PROGRAM PRG_IM2K4_PPM
VAR
    {attribute 'pytmc' := '
        pv: IM2K4:PPM
        io: io
    '}
    {attribute 'TcLinkTo' := '.fbGige.iIlluminatorINT := TIIB[IM2K4-EL4004-E7]^AO Outputs Channel 1^Analog output;
                              .fbGige.bGigePower := TIIB[IM2K4-EL2004-E3]^Channel 2^Output;
                              .fbPowerMeter.iVoltageINT := TIIB[IM2K4-EL3062-E6]^AI Standard Channel 1^Value;
                              .fbPowerMeter.fbThermoCouple.bError := TIIB[IM2K4-EL3314-E4]^TC Inputs Channel 1^Status^Error;
                              .fbPowerMeter.fbThermoCouple.bUnderrange := TIIB[IM2K4-EL3314-E4]^TC Inputs Channel 1^Status^Underrange;
                              .fbPowerMeter.fbThermoCouple.bOverrange := TIIB[IM2K4-EL3314-E4]^TC Inputs Channel 1^Status^Overrange;
                              .fbPowerMeter.fbThermoCouple.iRaw := TIIB[IM2K4-EL3314-E4]^TC Inputs Channel 1^Value;
                              .fbYagThermoCouple.bError := TIIB[IM2K4-EL3314-E4]^TC Inputs Channel 2^Status^Error;
                              .fbYagThermoCouple.bUnderrange := TIIB[IM2K4-EL3314-E4]^TC Inputs Channel 2^Status^Underrange;
                              .fbYagThermoCouple.bOverrange := TIIB[IM2K4-EL3314-E4]^TC Inputs Channel 2^Status^Overrange;
                              .fbYagThermoCouple.iRaw := TIIB[IM2K4-EL3314-E4]^TC Inputs Channel 2^Value'}
    fbIM2K4: FB_PPM;
END_VAR

fbIM2K4.nTransitionAssertionID := 16#2240;
fbIM2K4.nUnknownAssertionID := 16#2249;

fbIM2K4.stOut.fPosition := -8.59;
fbIM2K4.stOut.bUseRawCounts := FALSE;
fbIM2K4.stOut.nRequestAssertionID := 16#2241;
fbIM2K4.stOut.stBeamParams := PMPS_GVL.cstFullBeam;
fbIM2K4.stOut.bValid := TRUE;

fbIM2K4.stPower.fPosition := -47.69;
fbIM2K4.stPower.bUseRawCounts := FALSE;
fbIM2K4.stPower.nRequestAssertionID := 16#2242;
fbIM2K4.stPower.stBeamParams := PMPS_GVL.cstFullBeam;
fbIM2K4.stPower.bValid := TRUE;

fbIM2K4.stYag1.fPosition := -71.69;
fbIM2K4.stYag1.bUseRawCounts := FALSE;
fbIM2K4.stYag1.nRequestAssertionID := 16#2243;
fbIM2K4.stYag1.stBeamParams := PMPS_GVL.cstFullBeam;
fbIM2K4.stYag1.bValid := TRUE;

fbIM2K4.stYag2.fPosition := -97.70;
fbIM2K4.stYag2.bUseRawCounts := FALSE;
fbIM2K4.stYag2.nRequestAssertionID := 16#2244;
fbIM2K4.stYag2.stBeamParams := PMPS_GVL.cstFullBeam;
fbIM2K4.stYag2.bValid := TRUE;

fbIM2K4(
    fbArbiter := fbArbiter,
    fbFFHWO := fbFastFaultOutput1,
    stYStage := Main.M9);

END_PROGRAM

(* stored: Version 1.1.0.1, ProductVersion 3.1.4022.18
   POU PRG_IM2K4_PPM: Id {ba5f0424-d340-4eff-ab23-3e63bc2d0678}, SpecialFunc None *)
